// TwinCAT 3 PLC project PLC
// ProgramVersion: 3.1.4022.6
// libraries:
//   Tc2_MC2, * (Beckhoff Automation GmbH)
//   Tc2_NC, * (Beckhoff Automation GmbH)
//   Tc2_SPA, * (Beckhoff Automation GmbH)
//   Tc2_Standard, * (Beckhoff Automation GmbH)
//   Tc2_System, * (Beckhoff Automation GmbH)
//   Tc3_MC2_AdvancedHoming, * (Beckhoff Automation GmbH)
//   Tc3_Module, * (Beckhoff Automation GmbH)
//   VisuDialogs, * (System)
//   VisuSymbols, * (System)
//   BASIC,3.31,OSCAT
//   Visu Interfaces,newest,System
//   VisuElemEventTable,1.0.2.0,System
//   VisuElemsDateTime Interfaces,newest,Intern
//   VisuSymbols,3.5.10.0,System
// project tree:
//   DUTs/ dutInterlock.TcDUT
//   / GlobalTextList.TcGTLO, PlcTask.TcTTO, Visualization Manager.TcVMO (not stored), VISU_TASK.TcTTO
//   POUs/Cntrl/ progSCACntrl.TcPOU, progFCVCntrl.TcPOU, progHSVCntrl.TcPOU, progLITCntrl.TcPOU, progPITCntrl.TcPOU, progServoCntrl.TcPOU
//   POUs/FunctionBlocks/ fbFCV.TcPOU, fbHSV.TcPOU, fbPIT.TcPOU, fbLIT.TcPOU, fbSCA.TcPOU, fbServo.TcPOU
//   POUs/ MAIN.TcPOU
//   POUs/Simulation/ fbSimFCV.TcPOU, fbSimHSV.TcPOU, fbSimSCA.TcPOU
//   VISUs/Diag/FCV/ FCV_04_1001.TcVIS, FCV_04_1002.TcVIS, FCV_04_1003.TcVIS
//   VISUs/Diag/HSV/ HSV_04_1001.TcVIS, HSV_04_1002.TcVIS, HSV_04_1003.TcVIS, HSV_04_1004.TcVIS, HSV_04_1005.TcVIS
//   VISUs/Diag/SCA/ SCA_04_0100.TcVIS
//   VISUs/Screens/ Overview.TcVIS, Vacuum_C1.TcVIS (excluded from build)
//   VISUs/Templates/Diag/ visuFCVDiag.TcVIS, visuHSVDiag.TcVIS, visuLITDiag.TcVIS, visuPITDiag.TcVIS, visuSCADiag.TcVIS, visuTITDiag.TcVIS
//   VISUs/Templates/inDevelopment/ visuServoDiag.TcVIS
//   VISUs/Templates/Sym/ Vessel.TcVIS, visuHSVSim.TcVIS, visuFCVSim.TcVIS
//   VISUs/TrialAndError/ visu.TcVIS, Visualization.TcVIS
// real-time tasks:
//   TASK PlcTask: cycle T#10ms, priority 20, ADS port 350
//   TASK VISU_TASK: cycle T#200000us, priority 30, ADS port 351
// motion (NC):
//   TASK NC-Task 1 SAF: cycle T#2ms, priority 4, ADS port 501
//   TASK NC-Task 1 SVB: cycle T#10ms, priority 8, ADS port 511
//   AXIS Axis 1 (id 1)
//     OtherSettings: AllowMotionCmdToSlave=true
//     encoder EncType=1
//     drive DrvType=5
//       Analog: ScaleFactorActTorque=0.1
//       TimeComp: TaskDelayCycles=1
//     controller CtrType=1
//       CtrPara: PriorControlFactor=1
//         Observer: BandWidth=20
//   AXIS Axis 2 (id 2)
//     OtherSettings: AllowMotionCmdToSlave=true
//     encoder EncType=19
//       EncPara: MaxCount=#xffffffff
//     drive DrvType=16
//       DrvPara: MaxCount=#xffffffff
//         Analog: ScaleFactorActTorque=0.1
//         TimeComp: TaskDelayCycles=1
//     controller CtrType=1
//       CtrPara: PriorControlFactor=1
//         Observer: BandWidth=20

CONFIGURATION PLC
    RESOURCE PLC ON TwinCAT3
        TASK PlcTask(INTERVAL := T#10ms, PRIORITY := 20);
        TASK VISU_TASK(INTERVAL := T#200000us, PRIORITY := 30);
        PROGRAM MAIN WITH PlcTask : MAIN;
        PROGRAM VisuElems_Visu_Prg WITH VISU_TASK : VisuElems.Visu_Prg;
    END_RESOURCE
END_CONFIGURATION

// ---- DUTs/dutInterlock.TcDUT
TYPE dutInterlock :
STRUCT
	Intrlck_1 : BOOL;
	strIntrlck_1 : STRING;
	Intrlck_2 : BOOL;
	strIntrlck_2 : STRING;
	Intrlck_3 : BOOL;
	strIntrlck_3 : STRING;
	Intrlck_4 : BOOL;
	strIntrlck_4 : STRING;
	Intrlck_5 : BOOL;
	strIntrlck_5 : STRING;
	Intrlck_6 : BOOL;
	strIntrlck_6 : STRING;
	Intrlck_7 : BOOL;
	strIntrlck_7 : STRING;
	Intrlck_8 : BOOL;
	strIntrlck_8 : STRING;
	Intrlck_9 : BOOL;
	strIntrlck_9 : STRING;
	Intrlck_10 : BOOL;
	strIntrlck_10 : STRING;
	
	Intrlck_OK : BOOK;
	
END_STRUCT
END_TYPE

// ---- POUs/MAIN.TcPOU
PROGRAM MAIN
VAR
END_VAR

progHSVCntrl();
progFCVCntrl();
progLITCntrl();
progPITCntrl();
progSCACntrl();

END_PROGRAM

// ---- POUs/Cntrl/progHSVCntrl.TcPOU
PROGRAM progHSVCntrl
VAR
	HSV_04_0100 : fbHSV;

	HSV_04_1001 : fbHSV;
	HSV_04_1002 : fbHSV;
	HSV_04_1003 : fbHSV;
	HSV_04_1004 : fbHSV;
	HSV_04_1005 : fbHSV;
END_VAR

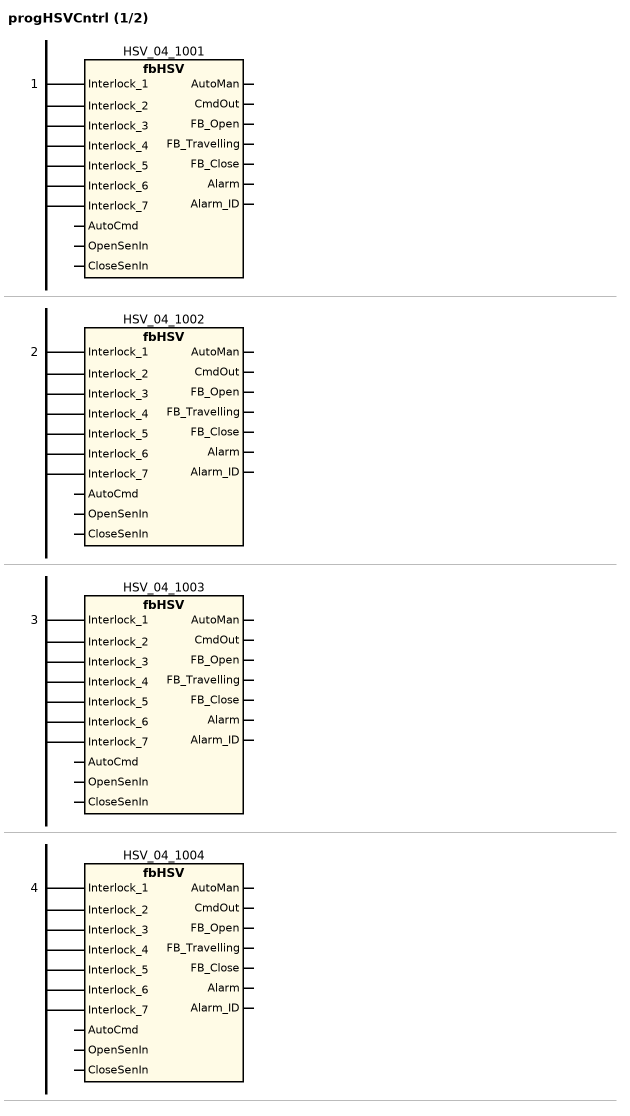
// NETWORK 1
HSV_04_1001(
    Interlock_1 := TRUE,
    Interlock_2 := TRUE,
    Interlock_3 := TRUE,
    Interlock_4 := TRUE,
    Interlock_5 := TRUE,
    Interlock_6 := TRUE,
    Interlock_7 := TRUE); // fbHSV

// NETWORK 2
HSV_04_1002(
    Interlock_1 := TRUE,
    Interlock_2 := TRUE,
    Interlock_3 := TRUE,
    Interlock_4 := TRUE,
    Interlock_5 := TRUE,
    Interlock_6 := TRUE,
    Interlock_7 := TRUE); // fbHSV

// NETWORK 3
HSV_04_1003(
    Interlock_1 := TRUE,
    Interlock_2 := TRUE,
    Interlock_3 := TRUE,
    Interlock_4 := TRUE,
    Interlock_5 := TRUE,
    Interlock_6 := TRUE,
    Interlock_7 := TRUE); // fbHSV

// NETWORK 4
HSV_04_1004(
    Interlock_1 := TRUE,
    Interlock_2 := TRUE,
    Interlock_3 := TRUE,
    Interlock_4 := TRUE,
    Interlock_5 := TRUE,
    Interlock_6 := TRUE,
    Interlock_7 := TRUE); // fbHSV

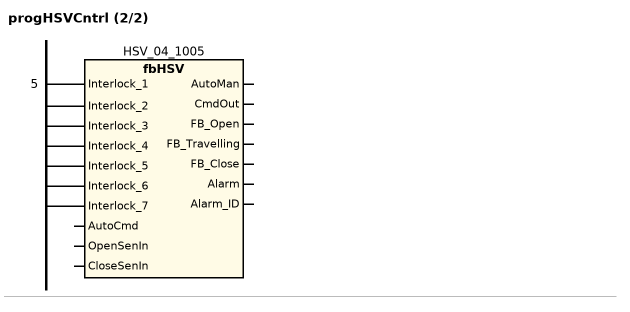
// NETWORK 5
HSV_04_1005(
    Interlock_1 := TRUE,
    Interlock_2 := TRUE,
    Interlock_3 := TRUE,
    Interlock_4 := TRUE,
    Interlock_5 := TRUE,
    Interlock_6 := TRUE,
    Interlock_7 := TRUE); // fbHSV

END_PROGRAM

// ---- POUs/FunctionBlocks/fbHSV.TcPOU
FUNCTION_BLOCK fbHSV
VAR_INPUT
	Interlock_1 : BOOL;
	Interlock_2 : BOOL;
	Interlock_3 : BOOL;
	Interlock_4 : BOOL;
	Interlock_5 : BOOL;
	Interlock_6 : BOOL;
	Interlock_7 : BOOL;

	AutoCmd : BOOL;
END_VAR
VAR_OUTPUT
	AutoMan : BOOL;
	FB_Open : BOOL;
	FB_Travelling : BOOL;
	FB_Close : BOOL;
	Alarm : BOOL;
	Alarm_ID : INT;
END_VAR
VAR
	CmdOut AT %Q* : BOOL;
	OpenSenIn AT %I*: BOOL;
	CloseSenIn AT %I* : BOOL;
	Interlock_OK : BOOL;
	AutoReq : BOOL;
	ManReq : BOOL;
	ManOpenReq : BOOL;
	ManCloseReq : BOOL;
	ManCmd : BOOL;
	strInterlock_1 : STRING;
	strInterlock_2 : STRING;
	strInterlock_3 : STRING;
	strInterlock_4 : STRING;
	strInterlock_5 : STRING;
	strInterlock_6 : STRING;
	strInterlock_7 : STRING;
	strAutoMan : STRING;
	strOpenTravClose : STRING;
	idxOpenTravClose : INT;
	EnableAlarm : BOOL;
	AlarmDelayTime : TIME := T#5S;
	tonAlarmDelay : TON;
	
	SimHSV : fbSimHSV;
END_VAR
VAR // added by the converter: edge detectors and wires of the graphical bodies
    _w1, _w2, _w3 : BOOL;
END_VAR

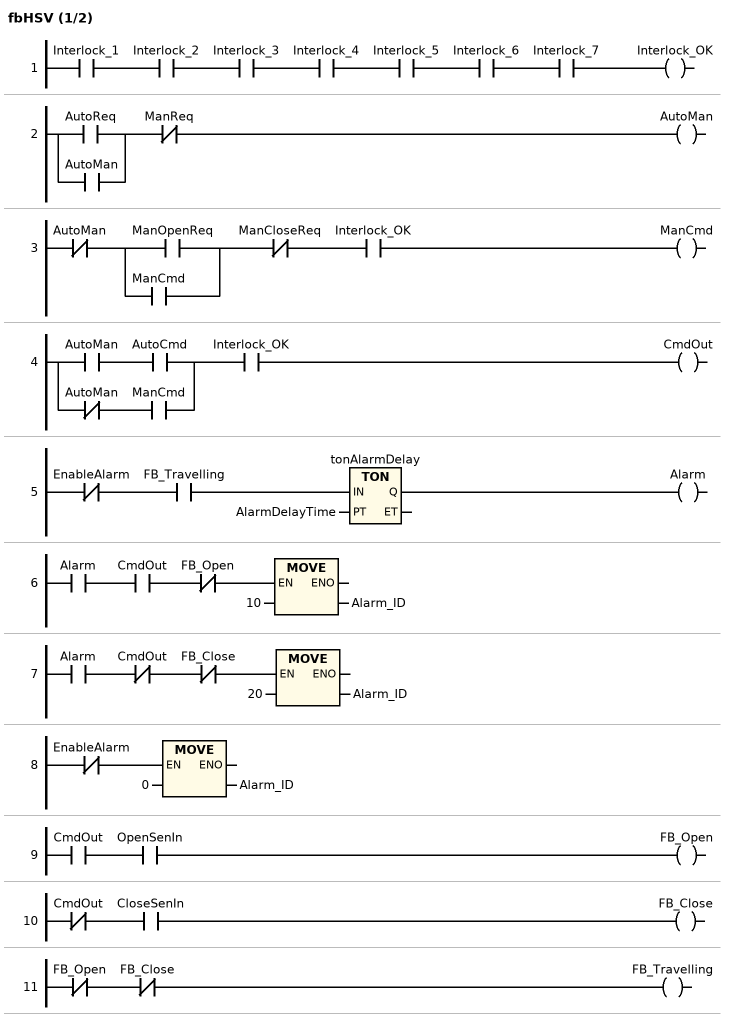
// NETWORK 1
Interlock_OK := Interlock_1 AND Interlock_2 AND Interlock_3 AND Interlock_4 AND Interlock_5 AND Interlock_6 AND Interlock_7;

// NETWORK 2
AutoMan := (AutoReq OR AutoMan) AND NOT ManReq;

// NETWORK 3
ManCmd := NOT AutoMan AND (ManOpenReq OR ManCmd) AND NOT ManCloseReq AND Interlock_OK;

// NETWORK 4
CmdOut := (AutoMan AND AutoCmd OR NOT AutoMan AND ManCmd) AND Interlock_OK;

// NETWORK 5
tonAlarmDelay(IN := NOT EnableAlarm AND FB_Travelling, PT := AlarmDelayTime); // TON
Alarm := tonAlarmDelay.Q;

// NETWORK 6
IF Alarm AND CmdOut AND NOT FB_Open THEN Alarm_ID := 10; END_IF

// NETWORK 7
IF Alarm AND NOT CmdOut AND NOT FB_Close THEN Alarm_ID := 20; END_IF

// NETWORK 8
IF NOT EnableAlarm THEN Alarm_ID := 0; END_IF

// NETWORK 9
FB_Open := CmdOut AND OpenSenIn;

// NETWORK 10
FB_Close := NOT CmdOut AND CloseSenIn;

// NETWORK 11
FB_Travelling := NOT FB_Open AND NOT FB_Close;

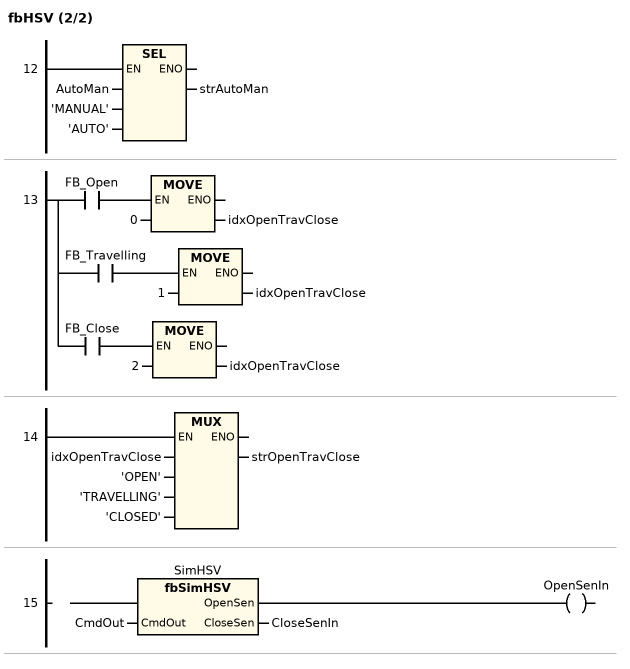
// NETWORK 12
strAutoMan := SEL(AutoMan, 'MANUAL', 'AUTO');

// NETWORK 13
_w1 := FB_Open;
IF _w1 THEN idxOpenTravClose := 0; END_IF
_w2 := FB_Travelling;
IF _w2 THEN idxOpenTravClose := 1; END_IF
_w3 := FB_Close;
IF _w3 THEN idxOpenTravClose := 2; END_IF
(* _w1 OR _w2 OR _w3; result not used *)

// NETWORK 14
strOpenTravClose := MUX(idxOpenTravClose, 'OPEN', 'TRAVELLING', 'CLOSED');

// NETWORK 15
SimHSV(CmdOut := CmdOut, CloseSen => CloseSenIn); // fbSimHSV
OpenSenIn := SimHSV.OpenSen;

END_FUNCTION_BLOCK

// ---- POUs/Simulation/fbSimHSV.TcPOU
FUNCTION_BLOCK fbSimHSV
VAR_INPUT
	CmdOut : BOOL;
END_VAR
VAR_OUTPUT
	OpenSen : BOOL;
	CloseSen : BOOL;
END_VAR
VAR
	tOpenning : TIME := T#50MS;
	tonOpenning : TON;
	tClosing : TIME := T#50MS;
	tonClosing : TON;
END_VAR

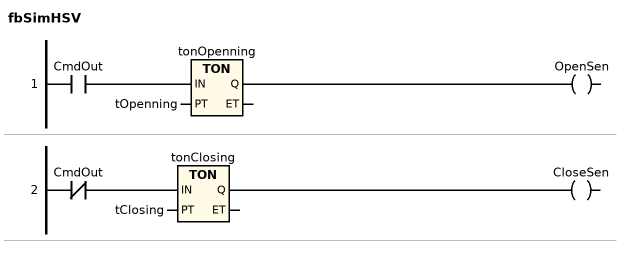
// NETWORK 1
tonOpenning(IN := CmdOut, PT := tOpenning); // TON
OpenSen := tonOpenning.Q;

// NETWORK 2
tonClosing(IN := NOT CmdOut, PT := tClosing); // TON
CloseSen := tonClosing.Q;

END_FUNCTION_BLOCK

// ---- POUs/Cntrl/progFCVCntrl.TcPOU
PROGRAM progFCVCntrl
VAR
	FCV_04_0100 : fbFCV;
	FCV_04_1001 : fbFCV;
	FCV_04_1002 : fbFCV;
	FCV_04_1003 : fbFCV;
END_VAR

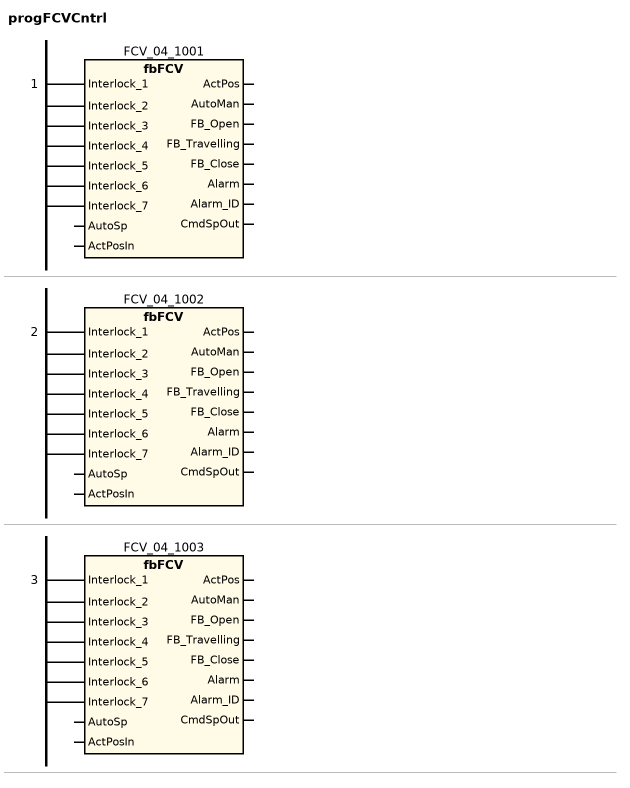
// NETWORK 1
FCV_04_1001(
    Interlock_1 := TRUE,
    Interlock_2 := TRUE,
    Interlock_3 := TRUE,
    Interlock_4 := TRUE,
    Interlock_5 := TRUE,
    Interlock_6 := TRUE,
    Interlock_7 := TRUE); // fbFCV

// NETWORK 2
FCV_04_1002(
    Interlock_1 := TRUE,
    Interlock_2 := TRUE,
    Interlock_3 := TRUE,
    Interlock_4 := TRUE,
    Interlock_5 := TRUE,
    Interlock_6 := TRUE,
    Interlock_7 := TRUE); // fbFCV

// NETWORK 3
FCV_04_1003(
    Interlock_1 := TRUE,
    Interlock_2 := TRUE,
    Interlock_3 := TRUE,
    Interlock_4 := TRUE,
    Interlock_5 := TRUE,
    Interlock_6 := TRUE,
    Interlock_7 := TRUE); // fbFCV

END_PROGRAM

// ---- POUs/FunctionBlocks/fbFCV.TcPOU
FUNCTION_BLOCK fbFCV
VAR_INPUT
	Interlock_1 : BOOL;
	Interlock_2 : BOOL;
	Interlock_3 : BOOL;
	Interlock_4 : BOOL;
	Interlock_5 : BOOL;
	Interlock_6 : BOOL;
	Interlock_7 : BOOL;

	AutoSp : REAL;
	ActPosIn : REAL;
END_VAR
VAR_OUTPUT
	ActPos : REAL;
	AutoMan : BOOL;
	FB_Open : BOOL;
	FB_Travelling : BOOL;
	FB_Close : BOOL;
	Alarm : BOOL;
	Alarm_ID : INT;

	CmdSpOut : REAL;
END_VAR
VAR
	Interlock_OK : BOOL;
	AutoReq : BOOL;
	ManReq : BOOL;
	ManSP : REAL;
	ManOpenReq : BOOL;
	ManCloseReq : BOOL;
	ManCmd : BOOL;
	rLowLimit : REAL;
	rLowLimitTol : REAL := 2;
	rHighLimit : REAL;
	rHighLimitTol : REAL := 2;

	strInterlock_1 : STRING;
	strInterlock_2 : STRING;
	strInterlock_3 : STRING;
	strInterlock_4 : STRING;
	strInterlock_5 : STRING;
	strInterlock_6 : STRING;
	strInterlock_7 : STRING;
	strAutoMan : STRING;
	strOpenTravClose : STRING;
	idxOpenTravClose : INT;
	EnableAlarm : BOOL;
	AlarmDelayTime : TIME := T#5S;
	tonAlarmDelay : TON;

	SimFCV : fbSimFCV;
END_VAR
VAR // added by the converter: edge detectors and wires of the graphical bodies
    _w1, _w2, _w3, _w4, _w5, _w6 : BOOL;
END_VAR

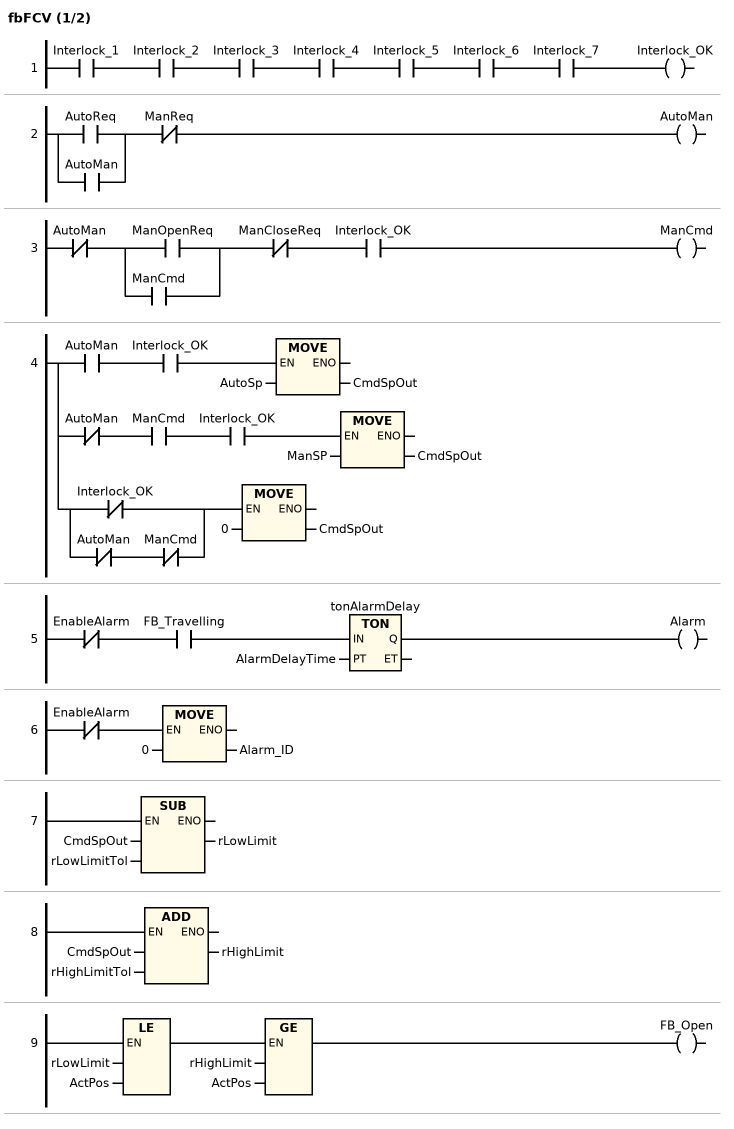
// NETWORK 1
Interlock_OK := Interlock_1 AND Interlock_2 AND Interlock_3 AND Interlock_4 AND Interlock_5 AND Interlock_6 AND Interlock_7;

// NETWORK 2
AutoMan := (AutoReq OR AutoMan) AND NOT ManReq;

// NETWORK 3
ManCmd := NOT AutoMan AND (ManOpenReq OR ManCmd) AND NOT ManCloseReq AND Interlock_OK;

// NETWORK 4
_w1 := AutoMan AND Interlock_OK;
IF _w1 THEN CmdSpOut := AutoSp; END_IF
_w2 := NOT AutoMan AND ManCmd AND Interlock_OK;
IF _w2 THEN CmdSpOut := ManSP; END_IF
_w3 := NOT Interlock_OK OR NOT AutoMan AND NOT ManCmd;
IF _w3 THEN CmdSpOut := 0; END_IF
(* _w1 OR _w2 OR _w3; result not used *)

// NETWORK 5
tonAlarmDelay(IN := NOT EnableAlarm AND FB_Travelling, PT := AlarmDelayTime); // TON
Alarm := tonAlarmDelay.Q;

// NETWORK 6
IF NOT EnableAlarm THEN Alarm_ID := 0; END_IF

// NETWORK 7
rLowLimit := CmdSpOut - rLowLimitTol;

// NETWORK 8
rHighLimit := CmdSpOut + rHighLimitTol;

// NETWORK 9
FB_Open := rLowLimit <= ActPos AND rHighLimit >= ActPos;

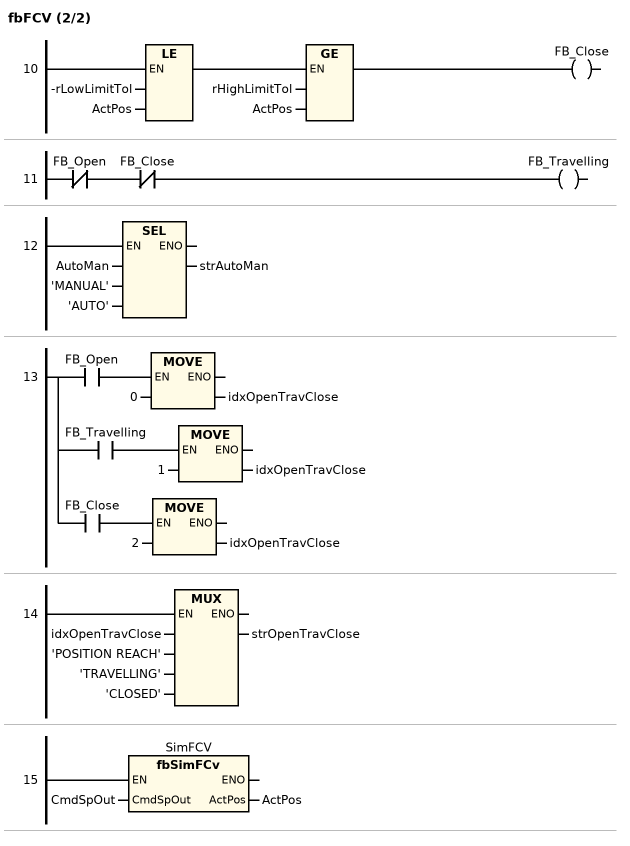
// NETWORK 10
FB_Close := (-rLowLimitTol) <= ActPos AND rHighLimitTol >= ActPos;

// NETWORK 11
FB_Travelling := NOT FB_Open AND NOT FB_Close;

// NETWORK 12
strAutoMan := SEL(AutoMan, 'MANUAL', 'AUTO');

// NETWORK 13
_w4 := FB_Open;
IF _w4 THEN idxOpenTravClose := 0; END_IF
_w5 := FB_Travelling;
IF _w5 THEN idxOpenTravClose := 1; END_IF
_w6 := FB_Close;
IF _w6 THEN idxOpenTravClose := 2; END_IF
(* _w4 OR _w5 OR _w6; result not used *)

// NETWORK 14
strOpenTravClose := MUX(idxOpenTravClose, 'POSITION REACH', 'TRAVELLING', 'CLOSED');

// NETWORK 15
SimFCV(CmdSpOut := CmdSpOut, ActPos => ActPos); // fbSimFCv

END_FUNCTION_BLOCK

// ---- POUs/Simulation/fbSimFCV.TcPOU
FUNCTION_BLOCK fbSimFCV
VAR_INPUT
	CmdSpOut : REAL;
END_VAR
VAR_OUTPUT
	ActPos : REAL;
END_VAR
VAR
	tonStepInc : TON;
	tStep : TIME := T#1MS;
	rStep : REAL := 1;
END_VAR

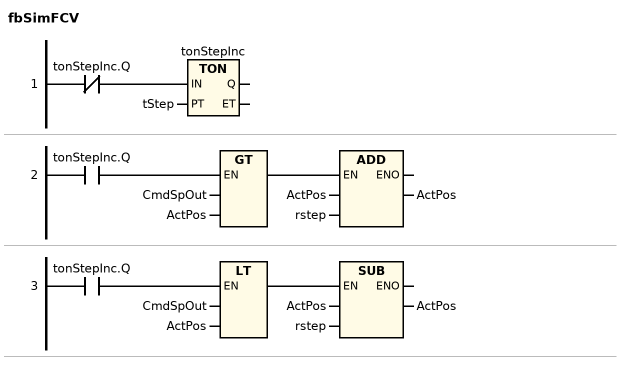
// NETWORK 1
tonStepInc(IN := NOT tonStepInc.Q, PT := tStep); // TON

// NETWORK 2
IF tonStepInc.Q AND CmdSpOut > ActPos THEN ActPos := ActPos + rstep; END_IF

// NETWORK 3
IF tonStepInc.Q AND CmdSpOut < ActPos THEN ActPos := ActPos - rstep; END_IF

END_FUNCTION_BLOCK

// ---- POUs/Cntrl/progLITCntrl.TcPOU
PROGRAM progLITCntrl
VAR
	LIT_04_0100 : fbLIT;
	
	LIT_04_1001 : fbLIT;
	LIT_04_1002 : fbLIT;
	LIT_04_1003 : fbLIT;

END_VAR

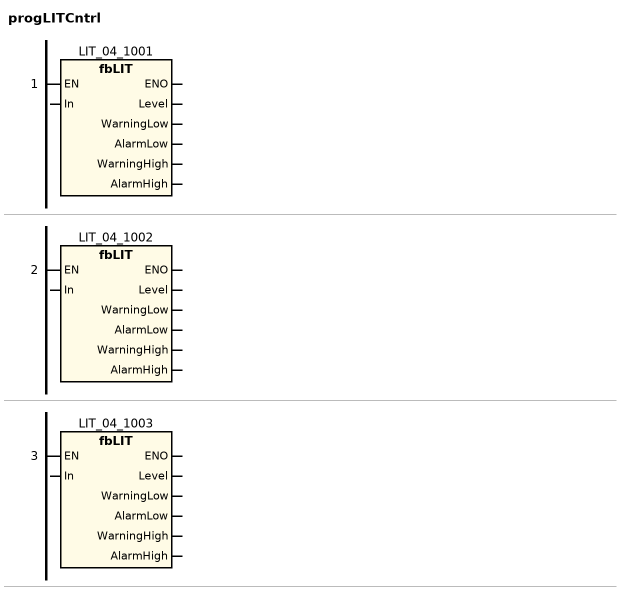
// NETWORK 1
LIT_04_1001(); // fbLIT

// NETWORK 2
LIT_04_1002(); // fbLIT

// NETWORK 3
LIT_04_1003(); // fbLIT

END_PROGRAM

// ---- POUs/FunctionBlocks/fbLIT.TcPOU
FUNCTION_BLOCK fbLIT
VAR_INPUT
	In : REAL;
END_VAR
VAR_OUTPUT
	Level : REAL;
	WarningLow : BOOL;
	AlarmLow : BOOL;
	WarningHigh : BOOL;
	AlarmHigh : BOOL;
END_VAR
VAR
	LLLimit : REAL := 10;
	LLimit : REAL := 20;
	HLimit : REAL := 80;
	HHLimit : REAL := 90;
	AlarmDelay : DINT := 10; // Alarm Delay in secondss
	HHDelayTON : TON;
	HDelayTON : TON;
	LDelayTON : TON;
	LLDelayTON : TON;
	tAlarmDelay: TIME;
END_VAR

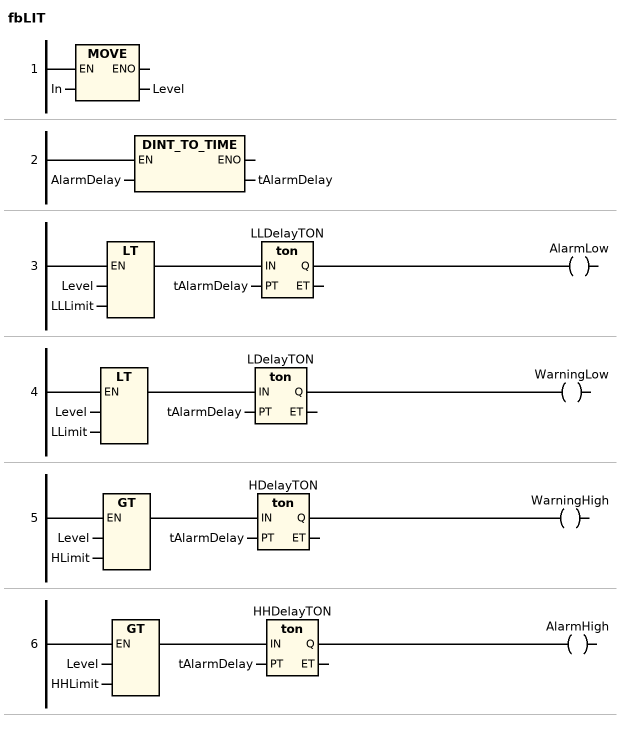
// NETWORK 1
Level := In;

// NETWORK 2
tAlarmDelay := DINT_TO_TIME(AlarmDelay);

// NETWORK 3
LLDelayTON(IN := Level < LLLimit, PT := tAlarmDelay); // ton
AlarmLow := LLDelayTON.Q;

// NETWORK 4
LDelayTON(IN := Level < LLimit, PT := tAlarmDelay); // ton
WarningLow := LDelayTON.Q;

// NETWORK 5
HDelayTON(IN := Level > HLimit, PT := tAlarmDelay); // ton
WarningHigh := HDelayTON.Q;

// NETWORK 6
HHDelayTON(IN := Level > HHLimit, PT := tAlarmDelay); // ton
AlarmHigh := HHDelayTON.Q;

END_FUNCTION_BLOCK

// ---- POUs/Cntrl/progPITCntrl.TcPOU
PROGRAM progPITCntrl
VAR
	PIT_04_0100 : fbPIT;
END_VAR

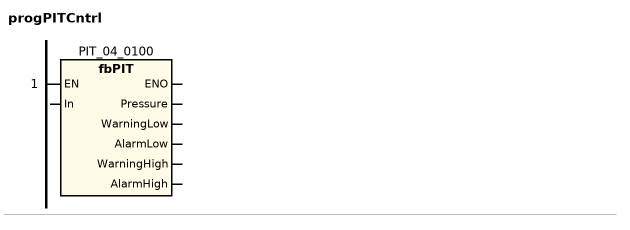
// NETWORK 1
PIT_04_0100(); // fbPIT

END_PROGRAM

// ---- POUs/FunctionBlocks/fbPIT.TcPOU
FUNCTION_BLOCK fbPIT
VAR_INPUT
	In : REAL;
END_VAR
VAR_OUTPUT
	Pressure : REAL;
	WarningLow : BOOL;
	AlarmLow : BOOL;
	WarningHigh : BOOL;
	AlarmHigh : BOOL;
END_VAR
VAR
	LLLimit : REAL := 10;
	LLimit : REAL := 20;
	HLimit : REAL := 80;
	HHLimit : REAL := 90;
	tDelayTime : TIME := T#0MS;
	tonAL : TON;
	tonWL : TON;
	tonWH : TON;
	tonAH : TON;
END_VAR

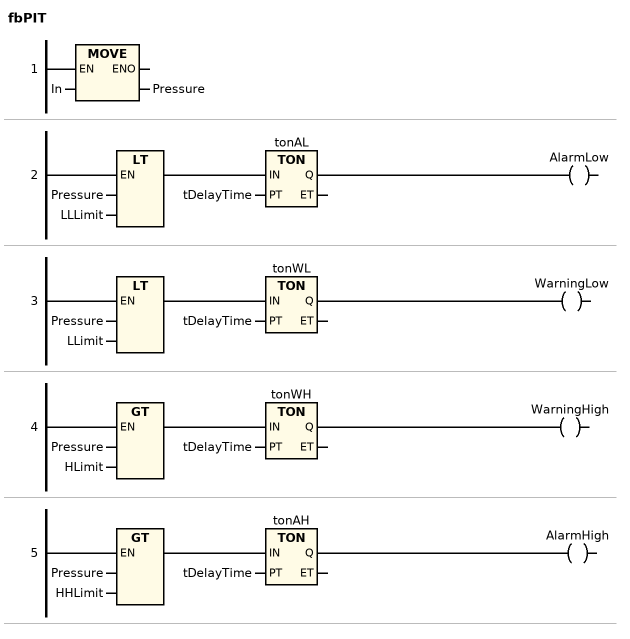
// NETWORK 1
Pressure := In;

// NETWORK 2
tonAL(IN := Pressure < LLLimit, PT := tDelayTime); // TON
AlarmLow := tonAL.Q;

// NETWORK 3
tonWL(IN := Pressure < LLimit, PT := tDelayTime); // TON
WarningLow := tonWL.Q;

// NETWORK 4
tonWH(IN := Pressure > HLimit, PT := tDelayTime); // TON
WarningHigh := tonWH.Q;

// NETWORK 5
tonAH(IN := Pressure > HHLimit, PT := tDelayTime); // TON
AlarmHigh := tonAH.Q;

END_FUNCTION_BLOCK

// ---- POUs/Cntrl/progSCACntrl.TcPOU
PROGRAM progSCACntrl
VAR
	Enable : BOOL;
	SCA_04_0100 : fbSCA;
END_VAR

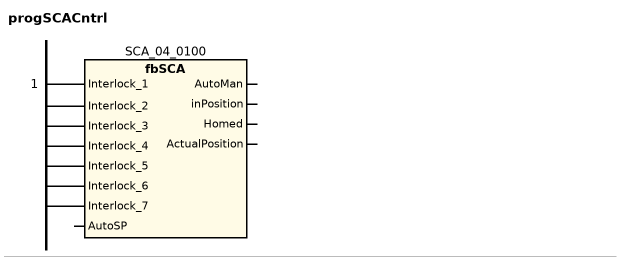
// NETWORK 1
SCA_04_0100(
    Interlock_1 := TRUE,
    Interlock_2 := TRUE,
    Interlock_3 := TRUE,
    Interlock_4 := TRUE,
    Interlock_5 := TRUE,
    Interlock_6 := TRUE,
    Interlock_7 := TRUE); // fbSCA

END_PROGRAM

// ---- POUs/FunctionBlocks/fbSCA.TcPOU
FUNCTION_BLOCK fbSCA
VAR_INPUT
	Interlock_1 : BOOL;
	Interlock_2 : BOOL;
	Interlock_3 : BOOL;
	Interlock_4 : BOOL;
	Interlock_5 : BOOL;
	Interlock_6 : BOOL;
	Interlock_7 : BOOL;
	
	AutoSP : REAL;
	CommandDirection : BOOL;
	AutoCmd : BOOL;
END_VAR
VAR_OUTPUT
	AutoMan : BOOL;
	ActualSpeed : REAL;
	ActualDirection : BOOL;
	Stopped : BOOL;
	Traveling : BOOL;
	Running : BOOL;
	Faulted : BOOL;
END_VAR
VAR
	StartCmdOut AT %Q* : BOOL;
	StopCmdOut AT %Q* : BOOL;
	Direction AT %Q* : BOOL;
	CommandSpeed : REAL;
	CommandSpeedRaw AT %Q* : DINT;
	ActualSpeedRaw AT %I*: DINT;
	Fault AT %I* : BOOL;
	EngMin : REAL := 0;		(* - means moving in the backward direction *)
	EngMax : REAL := 100;		(* the speed is expressed in percent *)
	RawMin : DINT := 2768;
	RawMax : DINT := 16535;
	Interlock_OK : BOOL;
	AutoReq : BOOL;
	ManReq : BOOL;
	ManSpeed : REAL;
	ManDirection : BOOL;
	ManStart : BOOL;
	ManStop : BOOL;

	strInterlock_1 : STRING;
	strInterlock_2 : STRING;
	strInterlock_3 : STRING;
	strInterlock_4 : STRING;
	strInterlock_5 : STRING;
	strInterlock_6 : STRING;
	strInterlock_7 : STRING;
	strAutoMan : STRING;
	idxStopTravRun : DINT;
	strStopTravRun : STRING;
	strOKFault : STRING;
	ClearFlt AT %Q* : BOOL;
	strAlmDesc : STRING;
	rCommandSpeed: REAL;		(* reserved variable *)
	
	simSCA : fbSimSCA;
	tmp: REAL;
END_VAR
VAR // added by the converter: edge detectors and wires of the graphical bodies
    _w1, _w2, _w3, _w4, _w5, _w6, _w7 : BOOL;
END_VAR

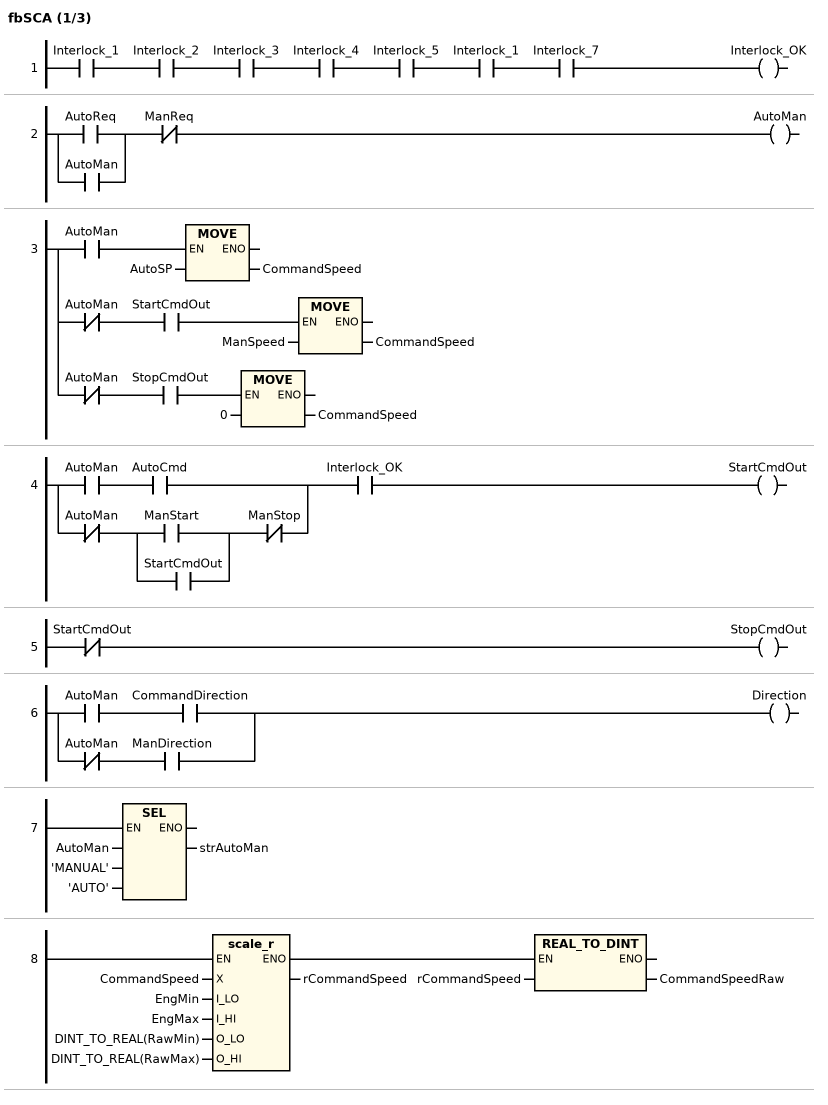
// NETWORK 1
Interlock_OK := Interlock_1 AND Interlock_2 AND Interlock_3 AND Interlock_4 AND Interlock_5 AND Interlock_1 AND Interlock_7;

// NETWORK 2
AutoMan := (AutoReq OR AutoMan) AND NOT ManReq;

// NETWORK 3
_w1 := AutoMan;
IF _w1 THEN CommandSpeed := AutoSP; END_IF
_w2 := NOT AutoMan AND StartCmdOut;
IF _w2 THEN CommandSpeed := ManSpeed; END_IF
_w3 := NOT AutoMan AND StopCmdOut;
IF _w3 THEN CommandSpeed := 0; END_IF
(* _w1 OR _w2 OR _w3; result not used *)

// NETWORK 4
StartCmdOut := (AutoMan AND AutoCmd OR NOT AutoMan AND (ManStart OR StartCmdOut) AND NOT ManStop) AND Interlock_OK;

// NETWORK 5
StopCmdOut := NOT StartCmdOut;

// NETWORK 6
Direction := AutoMan AND CommandDirection OR NOT AutoMan AND ManDirection;

// NETWORK 7
strAutoMan := SEL(AutoMan, 'MANUAL', 'AUTO');

// NETWORK 8
rCommandSpeed := scale_r(X := CommandSpeed, I_LO := EngMin, I_HI := EngMax, O_LO := DINT_TO_REAL(RawMin), O_HI := DINT_TO_REAL(RawMax));
CommandSpeedRaw := REAL_TO_DINT(rCommandSpeed);

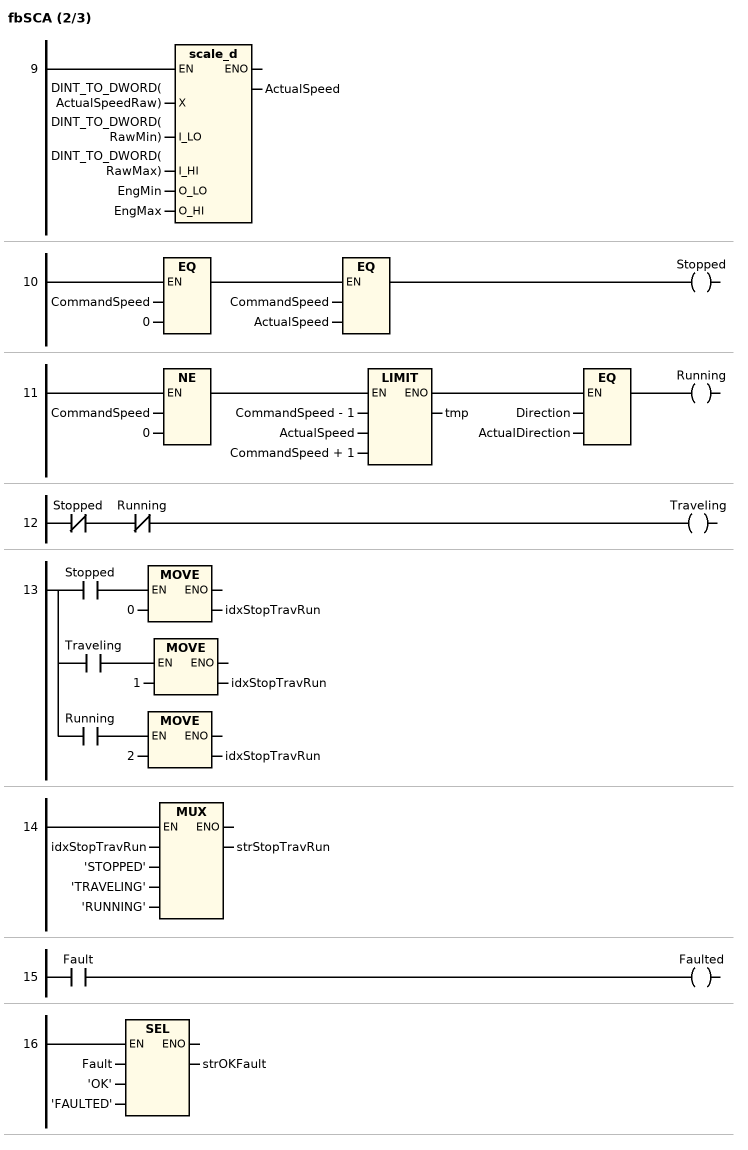
// NETWORK 9
ActualSpeed := scale_d(X := DINT_TO_DWORD(ActualSpeedRaw), I_LO := DINT_TO_DWORD(RawMin), I_HI := DINT_TO_DWORD(RawMax), O_LO := EngMin, O_HI := EngMax);

// NETWORK 10
Stopped := CommandSpeed = 0 AND CommandSpeed = ActualSpeed;

// NETWORK 11
_w4 := CommandSpeed <> 0;
IF _w4 THEN tmp := LIMIT(CommandSpeed - 1, ActualSpeed, CommandSpeed + 1); END_IF
Running := _w4 AND Direction = ActualDirection;

// NETWORK 12
Traveling := NOT Stopped AND NOT Running;

// NETWORK 13
_w5 := Stopped;
IF _w5 THEN idxStopTravRun := 0; END_IF
_w6 := Traveling;
IF _w6 THEN idxStopTravRun := 1; END_IF
_w7 := Running;
IF _w7 THEN idxStopTravRun := 2; END_IF
(* _w5 OR _w6 OR _w7; result not used *)

// NETWORK 14
strStopTravRun := MUX(idxStopTravRun, 'STOPPED', 'TRAVELING', 'RUNNING');

// NETWORK 15
Faulted := Fault;

// NETWORK 16
strOKFault := SEL(Fault, 'OK', 'FAULTED');

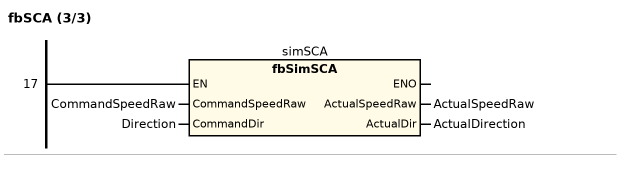
// NETWORK 17
simSCA(
    CommandSpeedRaw := CommandSpeedRaw,
    CommandDir := Direction,
    ActualSpeedRaw => ActualSpeedRaw,
    ActualDir => ActualDirection); // fbSimSCA

END_FUNCTION_BLOCK

// ---- POUs/Simulation/fbSimSCA.TcPOU
FUNCTION_BLOCK fbSimSCA
VAR_INPUT
	CommandSpeedRaw : DINT;
	CommandDir : BOOL; // 1 = Forward, 0 = Backward
END_VAR
VAR_OUTPUT
	ActualSpeedRaw : DINT;
	ActualDir : BOOL; // 1 = Forward, 0 = Backward
END_VAR
VAR
	Acceleration : DINT := 10; // defines the spead change per PLC cycle time
	CommandSpeed: DINT;
	ActualSpeed: DINT := 0;
END_VAR

IF CommandDir THEN
	CommandSpeed := CommandSpeedRaw;
ELSE
	CommandSpeed := -CommandSpeedRaw;
END_IF

IF ActualSpeed > 0 THEN
	ActualDir := 1;
	ActualSpeedRaw := ActualSpeed;
ELSE
	ActualDir := 0;
	ActualSpeedRaw := -ActualSpeed;
END_IF

IF ActualSpeed < CommandSpeed - Acceleration THEN
	ActualSpeed := ActualSpeed + Acceleration;
END_IF

IF ActualSpeed > CommandSpeed + Acceleration THEN
	ActualSpeed := ActualSpeed - Acceleration;
END_IF

IF ActualSpeed >= CommandSpeed - Acceleration AND ActualSpeed <= CommandSpeed + Acceleration THEN
	ActualSpeed := CommandSpeed;
END_IF

END_FUNCTION_BLOCK

// ---- POUs/Cntrl/progServoCntrl.TcPOU
PROGRAM progServoCntrl
VAR
	Servo_04_0100 : fbServo;
	
END_VAR

END_PROGRAM

// ---- POUs/FunctionBlocks/fbServo.TcPOU
FUNCTION_BLOCK fbServo
VAR_INPUT
	Interlock_1 : BOOL;
	Interlock_2 : BOOL;
	Interlock_3 : BOOL;
	Interlock_4 : BOOL;
	Interlock_5 : BOOL;
	Interlock_6 : BOOL;
	Interlock_7 : BOOL;

	AutoGoToPos : BOOL;
	Stop : BOOL;
	AutoPosSp : REAL;
	AutoSpeedSp : REAL; // % from max
	AutoAccSp : REAL; // % from max
	AutoJerkSp : REAL; // % from max
END_VAR
VAR_OUTPUT
	AutoMan : BOOL;
	PositionReached : BOOL;
	Running : BOOL;
	Faulted : BOOL;

	Position : REAL;
	Speed : REAL;
END_VAR
VAR
	Interlock_OK : BOOL;
	AutoReq : BOOL;
	ManReq : BOOL;

	ManPosSP : REAL;
	ManSpeedSP : REAL;
	ManAccSP : REAL;
	ManJerk : REAL;
	GoToPosition : BOOL;
	HomeReq : BOOL;
	JogForward : BOOL;
	JogBackward : BOOL;
	ClearFault : BOOL;
	FaultID : BOOL;
	
	PosSP : REAL;
	SpeedSP : REAL;
	AccSP : REAL;
	JerkSP : REAL;

	strInterlock_1 : STRING;
	strInterlock_2 : STRING;
	strInterlock_3 : STRING;
	strInterlock_4 : STRING;
	strInterlock_5 : STRING;
	strInterlock_6 : STRING;
	strInterlock_7 : STRING;
	strAutoMan : STRING;
END_VAR
VAR // added by the converter: edge detectors and wires of the graphical bodies
    _w1, _w2, _w3, _w4, _w5, _w6, _w7, _w8 : BOOL;
END_VAR

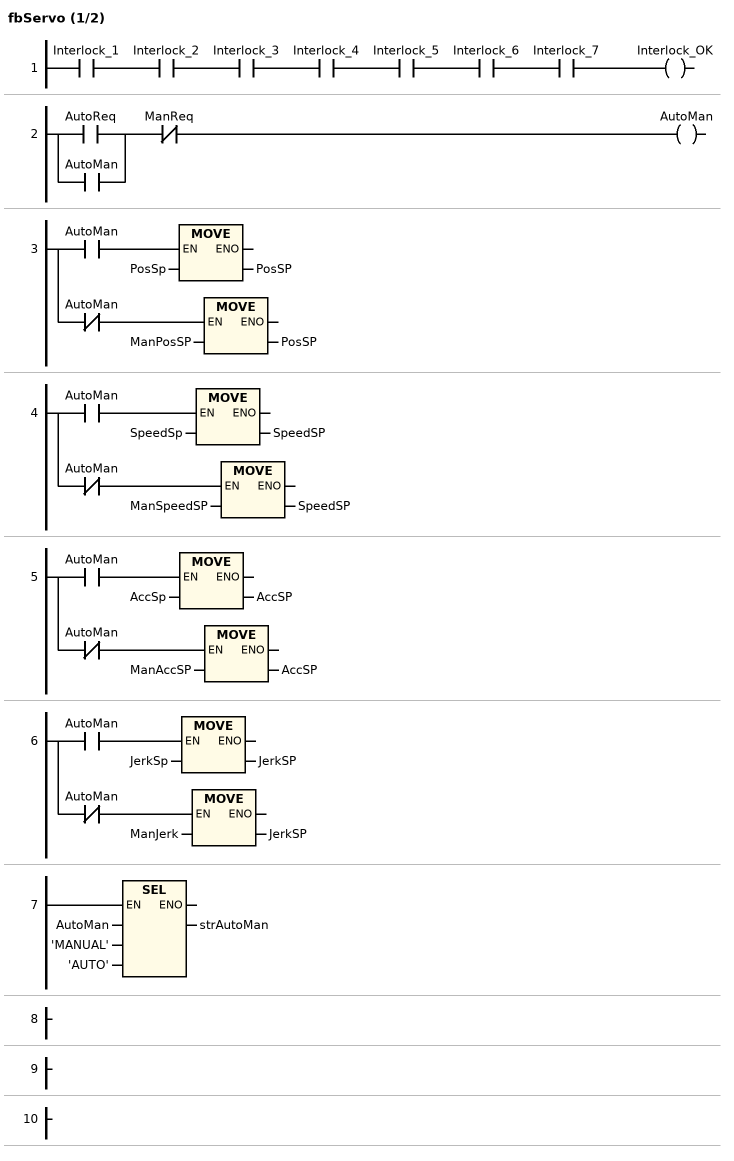
// NETWORK 1
Interlock_OK := Interlock_1 AND Interlock_2 AND Interlock_3 AND Interlock_4 AND Interlock_5 AND Interlock_6 AND Interlock_7;

// NETWORK 2
AutoMan := (AutoReq OR AutoMan) AND NOT ManReq;

// NETWORK 3
_w1 := AutoMan;
IF _w1 THEN PosSP := PosSp; END_IF
_w2 := NOT AutoMan;
IF _w2 THEN PosSP := ManPosSP; END_IF
(* _w1 OR _w2; result not used *)

// NETWORK 4
_w3 := AutoMan;
IF _w3 THEN SpeedSP := SpeedSp; END_IF
_w4 := NOT AutoMan;
IF _w4 THEN SpeedSP := ManSpeedSP; END_IF
(* _w3 OR _w4; result not used *)

// NETWORK 5
_w5 := AutoMan;
IF _w5 THEN AccSP := AccSp; END_IF
_w6 := NOT AutoMan;
IF _w6 THEN AccSP := ManAccSP; END_IF
(* _w5 OR _w6; result not used *)

// NETWORK 6
_w7 := AutoMan;
IF _w7 THEN JerkSP := JerkSp; END_IF
_w8 := NOT AutoMan;
IF _w8 THEN JerkSP := ManJerk; END_IF
(* _w7 OR _w8; result not used *)

// NETWORK 7
strAutoMan := SEL(AutoMan, 'MANUAL', 'AUTO');

// NETWORK 8

// NETWORK 9

// NETWORK 10

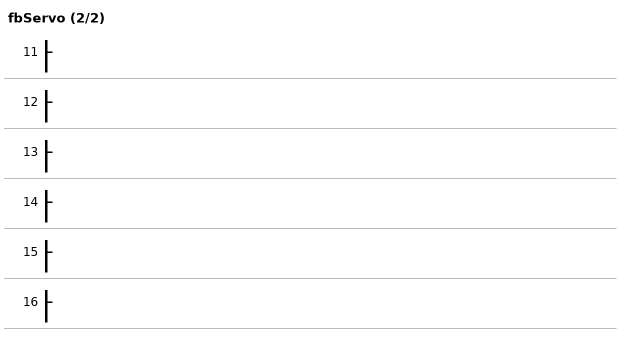
// NETWORK 11

// NETWORK 12

// NETWORK 13

// NETWORK 14

// NETWORK 15

// NETWORK 16

END_FUNCTION_BLOCK

// ---- GlobalTextList.TcGTLO
TEXTLIST GlobalTextList
  140 = '%'
  414 = '%3.2f'
  415 = '%3.2f %%'
  395 = '%3.2f mm'
  623 = '%d s'
  55 = '%s'
  498 = 'Acceleration'
  911 = 'Acknowledge' | English: 'Acknowledge'
  379 = 'Act'
  825 = 'Actual Level' | English: 'Actual Level' | Македонски: 'Моментално Ниво'
  210 = 'Actual position:' | English: 'Actual Position' | Македонски: 'Моментална Позиција'
  302 = 'Actual Presssure' | English: 'Actual Pressure' | Македонски: 'Моментален Притисок'
  769 = 'Actual set point:' | English: 'Actual Set Point' | Македонски: 'Моментален Сет Поинт'
  537 = 'Actual speed:' | English: 'Actual Speed' | Македонски: 'Моментална брзина'
  524 = 'Actual Temprature' | English: 'Actual Temperature' | Македонски: 'Моментална Температура'
  208 = 'Admin'
  311 = 'Alarm Delay Timer' | English: 'Alacm Delay Timer' | Македонски: 'Време на одложување'
  760 = 'Alarm High Limit' | English: 'Alarm High Limit' | Македонски: 'Аларм за високо ново'
  984 = 'Alarm Low Limit' | English: 'Alarm Low Limit' | Македонски: 'Аларм за ниско ниво'
  756 = 'AUTO' | English: 'Auto' | Македонски: 'Автоматски режим'
  23 = 'Auto'
  642 = 'Auto position set point'
  375 = 'Auto set point:' | English: 'Auto Set Point' | Македонски: 'Автоматски Сет Поинт'
  796 = 'BACKWARD' | English: 'Backward' | Македонски: 'Наназад'
  891 = 'Cancel' | English: 'Cancel' | Македонски: 'Исклучи'
  215 = 'CLEAR FAULT' | English: 'Clear Fault' | Македонски: 'Избриши Грешки'
  442 = 'CLOSE' | English: 'Close' | Македонски: 'Исклучи'
  975 = 'Enable' | English: 'Enable' | Македонски: 'Овозможи'
  144 = 'Enable Alarm' | English: 'Enable Alarm' | Македонски: 'Овозможи Аларм'
  277 = 'FORWARD' | English: 'Forward' | Македонски: 'Напред'
  172 = 'GO   TO   POSITION' | English: 'Go To Position' | Македонски: 'Оди на Позиција'
  515 = 'Go To Position'
  928 = 'HOME' | English: 'Home' | Македонски: 'Хомирај'
  394 = 'Home'
  80 = 'Jerk'
  247 = 'JOG   BACKWARD' | English: 'Jog Backward' | Македонски: 'Џогирај Назад'
  511 = 'JOG  FORWARD' | English: 'Jog Forward' | Македонски: 'Џогирај Напред'
  800 = 'Jog Backward'
  437 = 'Jog Forward'
  360 = 'Man'
  444 = 'MANUAL' | English: 'Manual' | Македонски: 'Рачен Режим'
  916 = 'Manual'
  418 = 'Manual position set point:'
  526 = 'Manual set point:' | English: 'Manual Set Point' | Македонски: 'Рачен Сет Поинт'
  881 = 'None'
  449 = 'OPEN' | English: 'Open' | Македонски: 'Отвори'
  598 = 'Operator'
  443 = 'Position'
  349 = 'Reverse' | English: 'Reverse' | Македонски: 'Назад'
  899 = 'REVERSE' | English: 'reverse' | Македонски: 'Назад'
  416 = 'SCA_04_0100'
  667 = 'SEMI AUTO'
  403 = 'Service'
  775 = 'Servo_04_0100'
  472 = 'Set Point:' | English: 'Set Point' | Македонски: 'Сет Поинт'
  635 = 'Speed'
  527 = 'START' | English: 'Start' | Македонски: 'Старт'
  562 = 'State'
  127 = 'STOP' | English: 'Stop' | Македонски: 'Стоп'
  424 = 'Warning High Limit' | English: 'Warning Hight Limit' | Македонски: 'Предупредување за Високо Ниво'
  417 = 'Warning Low Limit' | English: 'Warning Low Limit' | Македонски: 'Предупредување за Ниско Ниво'
END_TEXTLIST

// ---- VISUs/Diag/FCV/FCV_04_1001.TcVIS
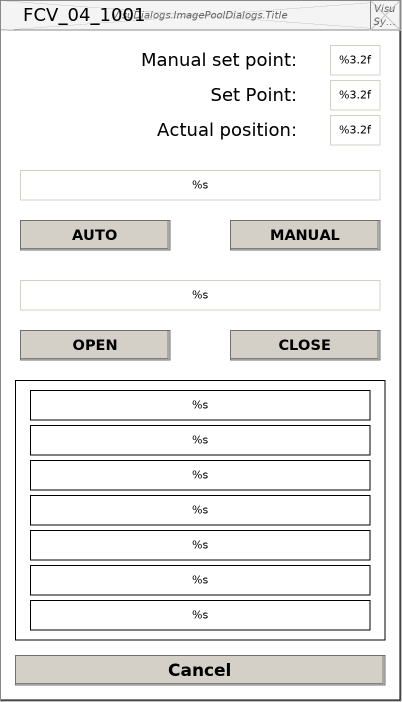
VISUALIZATION FCV_04_1001  // 402x702
    Rectangle (0,0 400x700)
    Button (20,220 150x30), "AUTO"
        tap progFCVCntrl.FCV_04_1001.AutoReq
    Button (230,220 150x30), "MANUAL"
        tap progFCVCntrl.FCV_04_1001.ManReq
    Button (20,330 150x30), "OPEN"
        tap progFCVCntrl.FCV_04_1001.ManOpenReq
    Button (230,330 150x30), "CLOSE"
        tap progFCVCntrl.FCV_04_1001.ManCloseReq
    Textfield (20,170 360x30), "%s", text variable: progFCVCntrl.FCV_04_1001.strAutoMan
    Textfield (20,280 360x30), "%s", text variable: progFCVCntrl.FCV_04_1001.strOpenTravClose
    Image (0,0 400x30), image: VisuDialogs.ImagePoolDialogs.Title
    Group (370,0 30x30)
        RoundedRectangle (0,0 30x30)
        Image (0,0 30x30), image: VisuSymbols.Symbols.Wrong
    Rectangle (15,380 370x260)
    RoundedRectangle (30,390 340x30), "%s", text variable: progFCVCntrl.FCV_04_1001.strInterlock_1
    RoundedRectangle (30,425 340x30), "%s", text variable: progFCVCntrl.FCV_04_1001.strInterlock_2
    RoundedRectangle (30,460 340x30), "%s", text variable: progFCVCntrl.FCV_04_1001.strInterlock_3
    RoundedRectangle (30,495 340x30), "%s", text variable: progFCVCntrl.FCV_04_1001.strInterlock_4
    RoundedRectangle (30,530 340x30), "%s", text variable: progFCVCntrl.FCV_04_1001.strInterlock_5
    RoundedRectangle (30,565 340x30), "%s", text variable: progFCVCntrl.FCV_04_1001.strInterlock_6
    RoundedRectangle (30,600 340x30), "%s", text variable: progFCVCntrl.FCV_04_1001.strInterlock_7
    Button (15,655 370x30), "Cancel"
    Label (0,80 300x30), "Set Point:"
    Textfield (330,80 50x30), "%3.2f", text variable: progFCVCntrl.FCV_04_1001.CmdSpOut
    Label (0,45 300x30), "Manual set point:"
    Textfield (330,45 50x30), "%3.2f", text variable: progFCVCntrl.FCV_04_1001.ManSP
        OnMouseClick: write progFCVCntrl.FCV_04_1001.ManSP via VisuDialogs.NumpadExtended
    Label (0,115 300x30), "Actual position:"
    Textfield (330,115 50x30), "%3.2f", text variable: progFCVCntrl.FCV_04_1001.ActPos
    Label (20,0 210x30), "FCV_04_1001"
END_VISUALIZATION

// ---- VISUs/Diag/FCV/FCV_04_1002.TcVIS
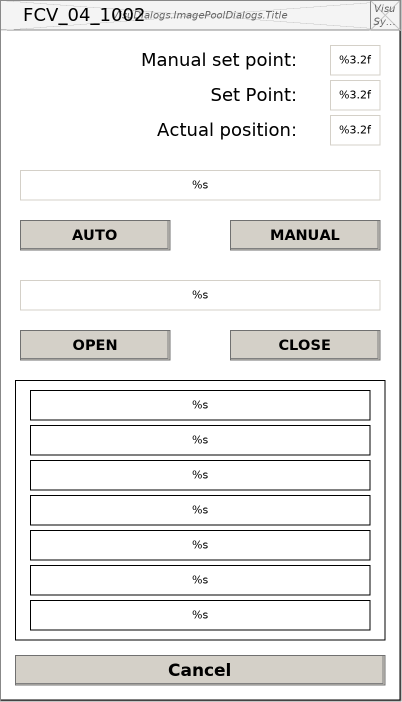
VISUALIZATION FCV_04_1002  // 402x702
    Rectangle (0,0 400x700)
    Button (20,220 150x30), "AUTO"
        tap progFCVCntrl.FCV_04_1002.AutoReq
    Button (230,220 150x30), "MANUAL"
        tap progFCVCntrl.FCV_04_1002.ManReq
    Button (20,330 150x30), "OPEN"
        tap progFCVCntrl.FCV_04_1002.ManOpenReq
    Button (230,330 150x30), "CLOSE"
        tap progFCVCntrl.FCV_04_1002.ManCloseReq
    Textfield (20,170 360x30), "%s", text variable: progFCVCntrl.FCV_04_1002.strAutoMan
    Textfield (20,280 360x30), "%s", text variable: progFCVCntrl.FCV_04_1002.strOpenTravClose
    Image (0,0 400x30), image: VisuDialogs.ImagePoolDialogs.Title
    Group (370,0 30x30)
        RoundedRectangle (0,0 30x30)
        Image (0,0 30x30), image: VisuSymbols.Symbols.Wrong
    Rectangle (15,380 370x260)
    RoundedRectangle (30,390 340x30), "%s", text variable: progFCVCntrl.FCV_04_1002.strInterlock_1
    RoundedRectangle (30,425 340x30), "%s", text variable: progFCVCntrl.FCV_04_1002.strInterlock_2
    RoundedRectangle (30,460 340x30), "%s", text variable: progFCVCntrl.FCV_04_1002.strInterlock_3
    RoundedRectangle (30,495 340x30), "%s", text variable: progFCVCntrl.FCV_04_1002.strInterlock_4
    RoundedRectangle (30,530 340x30), "%s", text variable: progFCVCntrl.FCV_04_1002.strInterlock_5
    RoundedRectangle (30,565 340x30), "%s", text variable: progFCVCntrl.FCV_04_1002.strInterlock_6
    RoundedRectangle (30,600 340x30), "%s", text variable: progFCVCntrl.FCV_04_1002.strInterlock_7
    Button (15,655 370x30), "Cancel"
    Label (0,80 300x30), "Set Point:"
    Textfield (330,80 50x30), "%3.2f", text variable: progFCVCntrl.FCV_04_1002.CmdSpOut
    Label (0,45 300x30), "Manual set point:"
    Textfield (330,45 50x30), "%3.2f", text variable: progFCVCntrl.FCV_04_1002.ManSP
        OnMouseClick: write progFCVCntrl.FCV_04_1002.ManSP via VisuDialogs.NumpadExtended
    Label (0,115 300x30), "Actual position:"
    Textfield (330,115 50x30), "%3.2f", text variable: progFCVCntrl.FCV_04_1002.ActPos
    Label (20,0 210x30), "FCV_04_1002"
END_VISUALIZATION

// ---- VISUs/Diag/FCV/FCV_04_1003.TcVIS
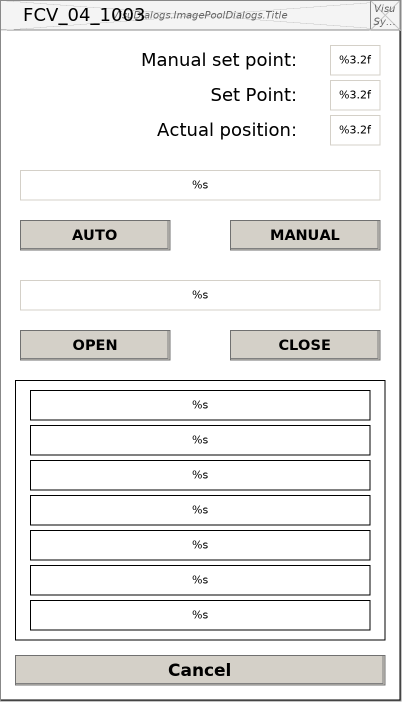
VISUALIZATION FCV_04_1003  // 402x702
    Rectangle (0,0 400x700)
    Button (20,220 150x30), "AUTO"
        tap progFCVCntrl.FCV_04_1003.AutoReq
    Button (230,220 150x30), "MANUAL"
        tap progFCVCntrl.FCV_04_1003.ManReq
    Button (20,330 150x30), "OPEN"
        tap progFCVCntrl.FCV_04_1003.ManOpenReq
    Button (230,330 150x30), "CLOSE"
        tap progFCVCntrl.FCV_04_1003.ManCloseReq
    Textfield (20,170 360x30), "%s", text variable: progFCVCntrl.FCV_04_1003.strAutoMan
    Textfield (20,280 360x30), "%s", text variable: progFCVCntrl.FCV_04_1003.strOpenTravClose
    Image (0,0 400x30), image: VisuDialogs.ImagePoolDialogs.Title
    Group (370,0 30x30)
        RoundedRectangle (0,0 30x30)
        Image (0,0 30x30), image: VisuSymbols.Symbols.Wrong
    Rectangle (15,380 370x260)
    RoundedRectangle (30,390 340x30), "%s", text variable: progFCVCntrl.FCV_04_1003.strInterlock_1
    RoundedRectangle (30,425 340x30), "%s", text variable: progFCVCntrl.FCV_04_1003.strInterlock_2
    RoundedRectangle (30,460 340x30), "%s", text variable: progFCVCntrl.FCV_04_1003.strInterlock_3
    RoundedRectangle (30,495 340x30), "%s", text variable: progFCVCntrl.FCV_04_1003.strInterlock_4
    RoundedRectangle (30,530 340x30), "%s", text variable: progFCVCntrl.FCV_04_1003.strInterlock_5
    RoundedRectangle (30,565 340x30), "%s", text variable: progFCVCntrl.FCV_04_1003.strInterlock_6
    RoundedRectangle (30,600 340x30), "%s", text variable: progFCVCntrl.FCV_04_1003.strInterlock_7
    Button (15,655 370x30), "Cancel"
    Label (0,80 300x30), "Set Point:"
    Textfield (330,80 50x30), "%3.2f", text variable: progFCVCntrl.FCV_04_1003.CmdSpOut
    Label (0,45 300x30), "Manual set point:"
    Textfield (330,45 50x30), "%3.2f", text variable: progFCVCntrl.FCV_04_1003.ManSP
        OnMouseClick: write progFCVCntrl.FCV_04_1003.ManSP via VisuDialogs.NumpadExtended
    Label (0,115 300x30), "Actual position:"
    Textfield (330,115 50x30), "%3.2f", text variable: progFCVCntrl.FCV_04_1003.ActPos
    Label (20,0 210x30), "FCV_04_1003"
END_VISUALIZATION

// ---- VISUs/Diag/HSV/HSV_04_1001.TcVIS
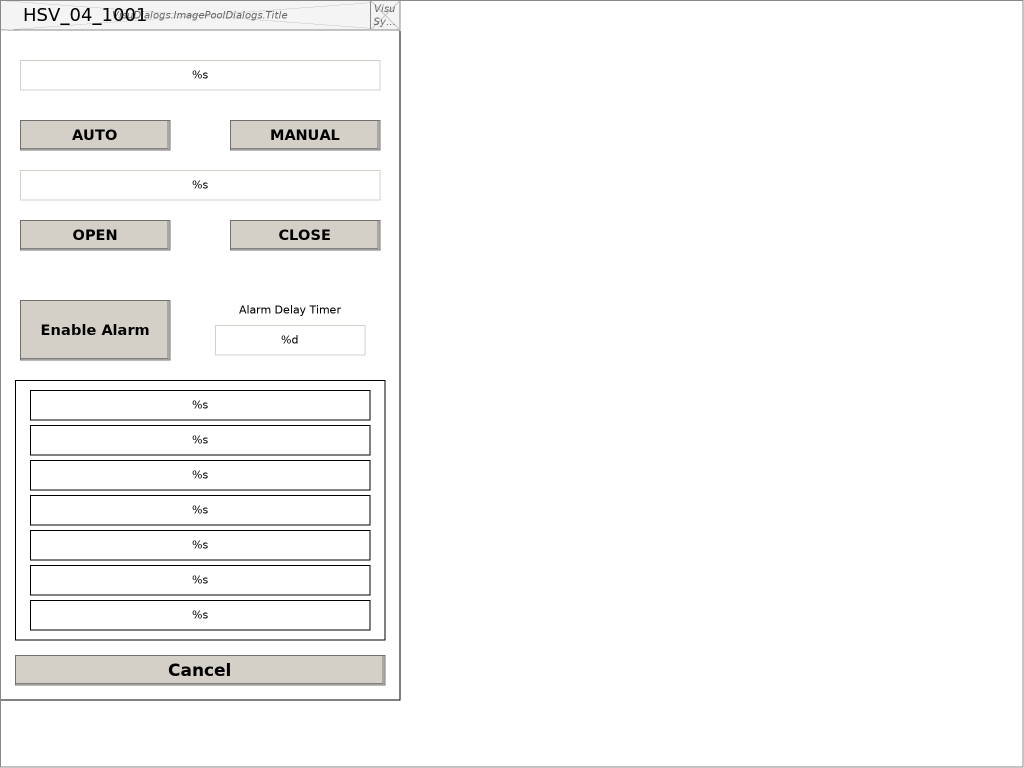
VISUALIZATION HSV_04_1001  // 1024x768
    Rectangle (0,0 400x700)
    Button (20,120 150x30), "AUTO"
        tap progHSVCntrl.HSV_04_1001.AutoReq
    Button (230,120 150x30), "MANUAL"
        tap progHSVCntrl.HSV_04_1001.ManReq
    Button (20,220 150x30), "OPEN"
        tap progHSVCntrl.HSV_04_1001.ManOpenReq
    Button (230,220 150x30), "CLOSE"
        tap progHSVCntrl.HSV_04_1001.ManCloseReq
    Textfield (20,60 360x30), "%s", text variable: progHSVCntrl.HSV_04_1001.strAutoMan
    Textfield (20,170 360x30), "%s", text variable: progHSVCntrl.HSV_04_1001.strOpenTravClose
    Button (20,300 150x60), "Enable Alarm"
        toggle progHSVCntrl.HSV_04_1001.EnableAlarm
    Textfield (215,325 150x30), "%d", text variable: progHSVCntrl.HSV_04_1001.AlarmDelayTime
    Label (215,295 150x30), "Alarm Delay Timer"
    Image (0,0 400x30), image: VisuDialogs.ImagePoolDialogs.Title
    Group (370,0 30x30)
        OnMouseClick: CloseDialog Dialog=HSV_04_1001, Result=OK, NumpadKeypadSet=True
        RoundedRectangle (0,0 30x30)
        Image (0,0 30x30), image: VisuSymbols.Symbols.Wrong
    Rectangle (15,380 370x260)
    RoundedRectangle (30,390 340x30), "%s", text variable: progHSVCntrl.HSV_04_1001.strInterlock_1
    RoundedRectangle (30,425 340x30), "%s", text variable: progHSVCntrl.HSV_04_1001.strInterlock_2
    RoundedRectangle (30,460 340x30), "%s", text variable: progHSVCntrl.HSV_04_1001.strInterlock_3
    RoundedRectangle (30,495 340x30), "%s", text variable: progHSVCntrl.HSV_04_1001.strInterlock_4
    RoundedRectangle (30,530 340x30), "%s", text variable: progHSVCntrl.HSV_04_1001.strInterlock_5
    RoundedRectangle (30,565 340x30), "%s", text variable: progHSVCntrl.HSV_04_1001.strInterlock_6
    RoundedRectangle (30,600 340x30), "%s", text variable: progHSVCntrl.HSV_04_1001.strInterlock_7
    Button (15,655 370x30), "Cancel"
        OnMouseClick: CloseDialog Dialog=HSV_04_1001, Result=OK, NumpadKeypadSet=True
    Label (20,0 210x30), "HSV_04_1001"
END_VISUALIZATION

// ---- VISUs/Diag/HSV/HSV_04_1002.TcVIS
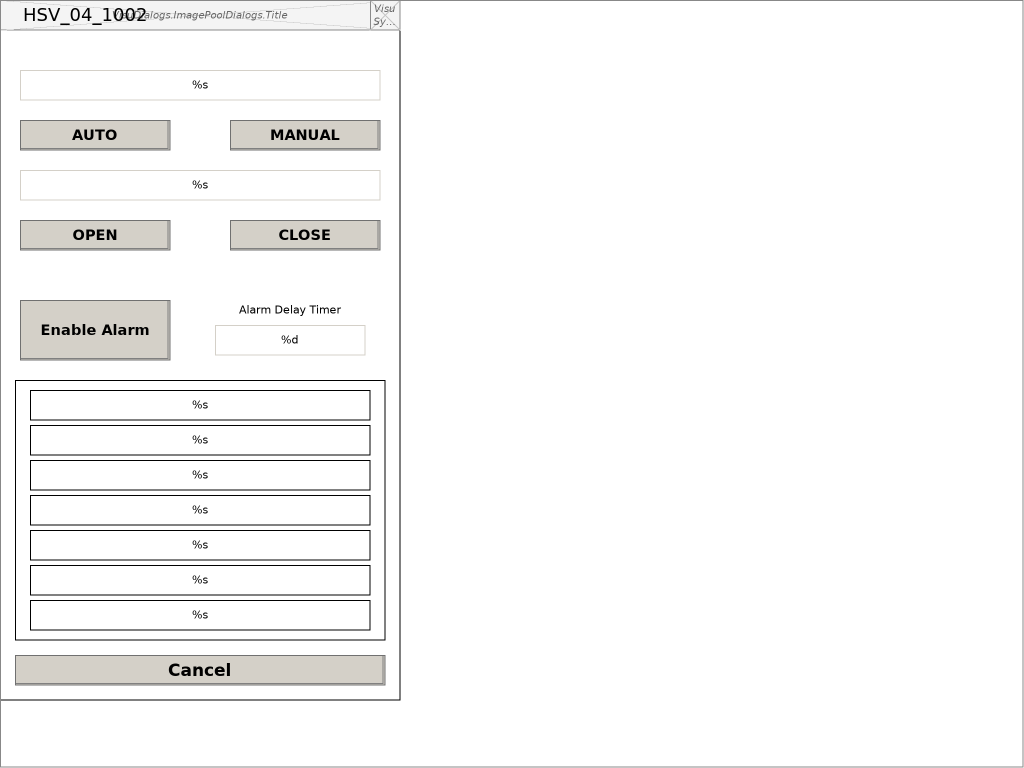
VISUALIZATION HSV_04_1002  // 1024x768
    Rectangle (0,0 400x700)
    Button (20,120 150x30), "AUTO"
        tap progHSVCntrl.HSV_04_1002.AutoReq
    Button (230,120 150x30), "MANUAL"
        tap progHSVCntrl.HSV_04_1002.ManReq
    Button (20,220 150x30), "OPEN"
        tap progHSVCntrl.HSV_04_1002.ManOpenReq
    Button (230,220 150x30), "CLOSE"
        tap progHSVCntrl.HSV_04_1002.ManCloseReq
    Textfield (20,70 360x30), "%s", text variable: progHSVCntrl.HSV_04_1002.strAutoMan
    Textfield (20,170 360x30), "%s", text variable: progHSVCntrl.HSV_04_1002.strOpenTravClose
    Button (20,300 150x60), "Enable Alarm"
        toggle progHSVCntrl.HSV_04_1002.EnableAlarm
    Textfield (215,325 150x30), "%d", text variable: progHSVCntrl.HSV_04_1002.AlarmDelayTime
    Label (215,295 150x30), "Alarm Delay Timer"
    Image (0,0 400x30), image: VisuDialogs.ImagePoolDialogs.Title
    Group (370,0 30x30)
        OnMouseClick: CloseDialog Dialog=HSV_04_1002, Result=OK, NumpadKeypadSet=True
        RoundedRectangle (0,0 30x30)
        Image (0,0 30x30), image: VisuSymbols.Symbols.Wrong
    Rectangle (15,380 370x260)
    RoundedRectangle (30,390 340x30), "%s", text variable: progHSVCntrl.HSV_04_1002.strInterlock_1
    RoundedRectangle (30,425 340x30), "%s", text variable: progHSVCntrl.HSV_04_1002.strInterlock_2
    RoundedRectangle (30,460 340x30), "%s", text variable: progHSVCntrl.HSV_04_1002.strInterlock_3
    RoundedRectangle (30,495 340x30), "%s", text variable: progHSVCntrl.HSV_04_1002.strInterlock_4
    RoundedRectangle (30,530 340x30), "%s", text variable: progHSVCntrl.HSV_04_1002.strInterlock_5
    RoundedRectangle (30,565 340x30), "%s", text variable: progHSVCntrl.HSV_04_1002.strInterlock_6
    RoundedRectangle (30,600 340x30), "%s", text variable: progHSVCntrl.HSV_04_1002.strInterlock_7
    Button (15,655 370x30), "Cancel"
        OnMouseClick: CloseDialog Dialog=HSV_04_1002, Result=OK, NumpadKeypadSet=True
    Label (20,0 210x30), "HSV_04_1002"
END_VISUALIZATION

// ---- VISUs/Diag/HSV/HSV_04_1003.TcVIS
